// Mitsubishi GX Works2 project: FX3U_生益PP   PLC: FX3U/FX3UC

PROGRAM MAIN
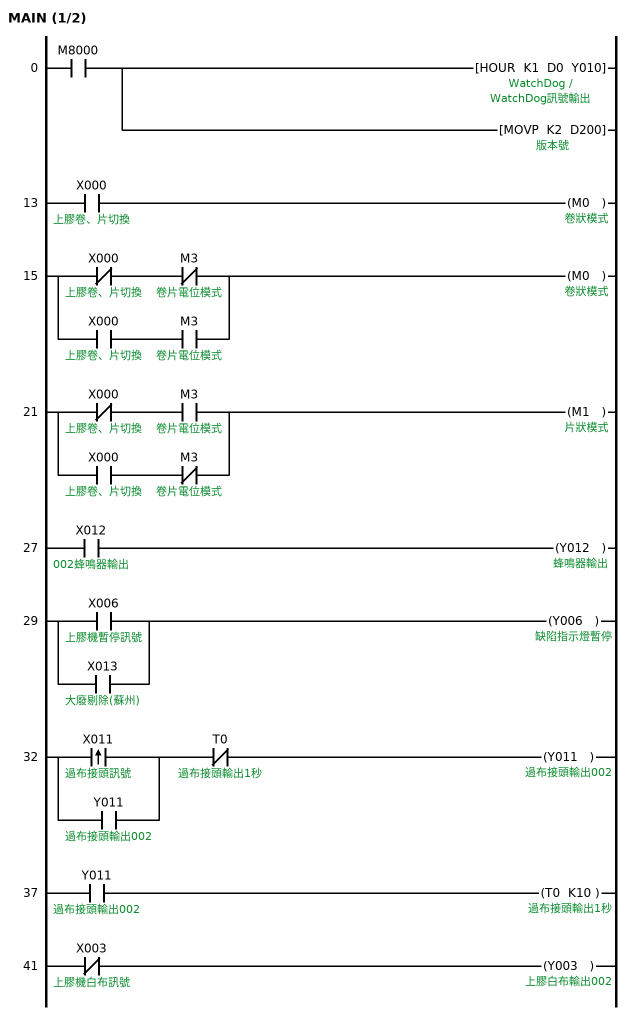
0     LD      M8000
      HOUR    K1 D0 Y010  ; WatchDog / WatchDog訊號輸出
      MOVP    K2 D200  ; 版本號
13    LD      X000  ; 上膠卷、片切換
      OUT     M0  ; 卷狀模式
15    LDI     X000  ; 上膠卷、片切換
      ANI     M3  ; 卷片電位模式
      LD      X000  ; 上膠卷、片切換
      AND     M3  ; 卷片電位模式
      ORB
      OUT     M0  ; 卷狀模式
21    LDI     X000  ; 上膠卷、片切換
      AND     M3  ; 卷片電位模式
      LD      X000  ; 上膠卷、片切換
      ANI     M3  ; 卷片電位模式
      ORB
      OUT     M1  ; 片狀模式
27    LD      X012  ; 002蜂鳴器輸出
      OUT     Y012  ; 蜂鳴器輸出
29    LD      X006  ; 上膠機暫停訊號
      OR      X013  ; 大廢剔除(蘇州)
      OUT     Y006  ; 缺陷指示燈暫停
32    LDP     X011  ; 過布接頭訊號
      OR      Y011  ; 過布接頭輸出002
      ANI     T0  ; 過布接頭輸出1秒
      OUT     Y011  ; 過布接頭輸出002
37    LD      Y011  ; 過布接頭輸出002
      OUT     T0 K10  ; 過布接頭輸出1秒
41    LDI     X003  ; 上膠機白布訊號
      OUT     Y003  ; 上膠白布輸出002
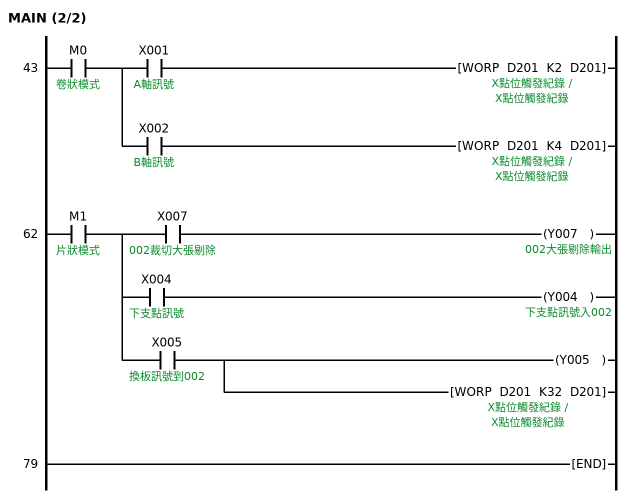
43    LD      M0  ; 卷狀模式
      MPS
      AND     X001  ; A軸訊號
      WORP    D201 K2 D201  ; X點位觸發紀錄
      MPP
      AND     X002  ; B軸訊號
      WORP    D201 K4 D201
62    LD      M1  ; 片狀模式
      MPS
      AND     X007  ; 002裁切大張剔除
      OUT     Y007  ; 002大張剔除輸出
      MRD
      AND     X004  ; 下支點訊號
      OUT     Y004  ; 下支點訊號入002
      MPP
      AND     X005  ; 換板訊號到002
      OUT     Y005
      WORP    D201 K32 D201
79    END
END_PROGRAM

// device comments not shown above
X010  ; WathDog(移除)
X017  ; 生益蘇州AB軸訊號
D1  ; WatchDog
D202  ; X點位觸發紀錄
